FUNCTION TryConvert_BOOL_TO_WORD : BOOL
VAR_INPUT
	in : BOOL;
	out : REFERENCE TO WORD;
END_VAR

out := BOOL_TO_WORD(in);
TryConvert_BOOL_TO_WORD := TRUE;

END_FUNCTION

(* stored: Version 1.1.0.1, ProductVersion 3.1.4024.12
   POU TryConvert_BOOL_TO_WORD: Id {07619fe8-6cb7-4d80-a5e9-db0289eaccc0}, SpecialFunc None *)
